TYPE DUT_PARAMETER_OUTPUT :
STRUCT
	///Free to use = TRUE, busy to use =FALSE
	Dummy: BOOL := TRUE;
	///ID of the parameter
	ID: UINT;
	///Name of the parameter
	Name: STRING(80);
	///Unit of the parameter
	Unit: STRING(80);
	///Optional parameter
	Required: BOOL;
	///Default parameter to work
	Default: LREAL;
	///Minimum value of the parameter
	MinValue: LREAL;
	///Maximum value of the parameter
	MaxValue: LREAL;
END_STRUCT
END_TYPE

(* stored: Version 1.1.0.1, ProductVersion 3.1.0.25
   DUT DUT_PARAMETER_OUTPUT: Id {6c781562-b4ad-4713-8e7c-601b4930d059} *)
